FUNCTION_BLOCK TestType
  (* Version 1.0, 2005-04-08, Goran Cengic, Chalmers *)
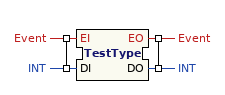
  EVENT_INPUT
    EI WITH DI;
  END_EVENT
  EVENT_OUTPUT
    EO WITH DO;
  END_EVENT
  VAR_INPUT
    DI : INT;
  END_VAR
  VAR_OUTPUT
    DO : INT;
  END_VAR
  VAR
    invoked : INT;
  END_VAR
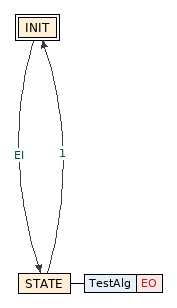
  EC_STATES
    INIT;
    STATE : TestAlg -> EO;
  END_STATES
  EC_TRANSITIONS
    INIT TO STATE := EI;
    STATE TO INIT := 1;
  END_TRANSITIONS
  ALGORITHM TestAlg IN Java:
invoked = (invoked + 1) % 3;
	DO = (DI + 1) % 3;
  END_ALGORITHM
END_FUNCTION_BLOCK
(* other elements stored in the file *)
(* ECAction Algorithm="PrintAlg"/ *)
(* Algorithm Name="PrintAlg"> <Other Language="Java" Text= "System.out.println(&#34;TestAlg:invoked: &#34; + invoked + &#34; times.&#34;); System.out.println(&#34;TestAlg: DO: &#34; + DO + &#34;.&#34;);" /> </Algorithm *)
